{attribute 'qualified_only'}
VAR_GLOBAL
END_VAR

(* stored: Version 1.1.0.1, ProductVersion 3.1.4020.12
   GVL StepperGVLs: Id {9c8a511a-1b4f-4744-88b0-142d0cb0514f} *)
